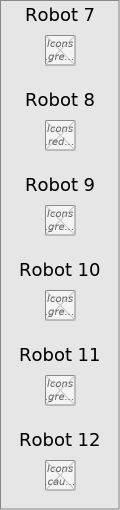
VISUALIZATION RightRobotStatus  // 120x510
    Textfield (0,0 120x30), "Robot 7"
    Textfield (0,85 120x30), "Robot 8"
    Textfield (0,170 120x30), "Robot 9"
    Textfield (0,255 120x30), "Robot 10"
    Textfield (0,340 120x30), "Robot 11"
    Textfield (0,425 120x30), "Robot 12"
    Image (45,35 30x30), input disabled if: TRUE, image: Icons.green-checkmark-icon
    Image (45,120 30x30), colour toggle: TRUE, input disabled if: TRUE, image: Icons.red-x-icon
    Image (45,205 30x30), input disabled if: TRUE, image: Icons.green-checkmark-icon
    Image (45,290 30x30), input disabled if: TRUE, image: Icons.green-checkmark-icon
    Image (45,375 30x30), input disabled if: TRUE, image: Icons.green-checkmark-icon
    Image (45,460 30x30), input disabled if: TRUE, image: Icons.caution-icon
        OnMouseClick: OpenDialog Dialog=VisuDialogs.MessageBox, Parameters={eType: , sMessageTxt: 'Warning Message Here', sTitle: 'WARNING'}, OpenModal=True, PositionX=312, PositionY=100
END_VISUALIZATION

(* stored: Version 1.1.0.1, ProductVersion 3.1.4024.15
   Visu RightRobotStatus: Id {98de1c2c-7432-4eef-8900-0fe81bc6fb03} *)
